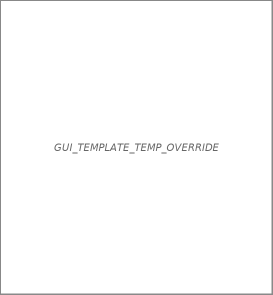
VISUALIZATION GUI_T2_OVERRIDE  // 273x295
    Frame (0,0 273x295)
        shows GUI_TEMPLATE_TEMP_OVERRIDE(m_Cmd := MAIN.tempOR_T2, m_Temp := MAIN.T2)
END_VISUALIZATION

(* stored: Version 1.1.0.1, ProductVersion 3.1.4024.12
   Visu GUI_T2_OVERRIDE: Id {5a87b174-2d4b-4595-b60e-2027be4f3336} *)
